PROGRAM MAIN
VAR
	//Main Terminal INPUTS
		//Part 1(Conveyor 1)	
	Inp_Part_at_Conveyor_1								AT%I*: BOOL;
	Inp_Plunger_Parts_Container_In						AT%I*: BOOL;
	Inp_Plunger_Parts_Container_Out						AT%I*: BOOL;
	Inp_Part_On_Conveyor_1								AT%I*: BOOL;
	Inp_Part_in_front_of_Parts_Alignment				AT%I*: BOOL;
	Inp_Plunger_Parts_Alignment_Left_In					AT%I*: BOOL;
	Inp_Plunger_Parts_Alignment_Left_Out				AT%I*: BOOL;
	Inp_Plunger_Parts_Alignment_Right_In				AT%I*: BOOL;	
	
	Inp_Plunger_Parts_Alignment_Right_Out				AT%I*: BOOL;
	Inp_Plunger_Parts_Alignment_Above_In				AT%I*: BOOL;
	Inp_Plunger_Parts_Alignment_Above_Out				AT%I*: BOOL;
	Inp_Part_in_front_of_Crane							AT%I*: BOOL;
	Inp_Crane_In										AT%I*: BOOL;
	Inp_Crane_Out										AT%I*: BOOL;
	Inp_Crane_Above										AT%I*: BOOL;
	Inp_Crane_Below										AT%I*: BOOL;
	
	Inp_Motor_1_Protection_Switch_is_OK					AT%I*: BOOL;
	Inp_Base_Positions									AT%I*: BOOL;
	Inp_Start_Button									AT%I*: BOOL;
	Inp_Stop_Button										AT%I*: BOOL;
	
		//Part 2(Conveyor 2)	
	Inp_Conveyor_2_Palette_Left_Side					AT%I*: BOOL;
	Inp_Conveyor_2_Palette_Right_Side					AT%I*: BOOL;
	Inp_Palette_in_front_of_Tester						AT%I*: BOOL;
	Inp_Stopper_Below									AT%I*: BOOL;
	Inp_Stopper_Above									AT%I*: BOOL;
	Inp_Feedback_from_Tester							AT%I*: BOOL;
	Inp_Reserve_1										AT%I*: BOOL;
	Inp_Motor_2_Protection_Switch_is_OK					AT%I*: BOOL;
	
	Inp_Conveyor_2_Pallete_Slider_In					AT%I*: BOOL;
	Inp_Conveyor_2_Pallete_Slider_Out					AT%I*: BOOL;
	Inp_Feedback_from_Tester_GOOD_Part					AT%I*: BOOL;
	Inp_Feedback_from_Tester_BAD_Part					AT%I*: BOOL;
		
		//Part 3(Conveyor 3)
	Inp_Conveyor_3_Palette_Left_Side					AT%I*: BOOL;
	Inp_Conveyor_3_Palette_Right_Side					AT%I*: BOOL;	
	Inp_Conveyor_3_Pallete_Slider_In					AT%I*: BOOL;
	Inp_Conveyor_3_Pallete_Slider_Out					AT%I*: BOOL;	
	Inp_Motor_3_Protection_Switch_is_OK					AT%I*: BOOL;

	//Coupler	
		//Part 4(Sorting System)
	Inp_Sorter_in_Basik_Position						AT%I*: BOOL;
	Inp_Sorter_Plunger_Above							AT%I*: BOOL;
	Inp_Sorter_Plunger_Below							AT%I*: BOOL;
	Inp_Measuring_Bar_Sorting_Axis_X					AT%I*: INT;
	Inp_Measuring_Bar_Sorting_Axis_Y					AT%I*: INT;
	Inp_Form_is_Changed_Button							AT%I*: BOOL;
	

	//Main Terminal OUTPUTS
		//Part 1(Conveyor 1)	
	Out_Conveyor_1_Motor_On								AT%Q*: BOOL;
	Out_Plunger_Parts_Container_Drive_In				AT%Q*: BOOL;
	Out_Plunger_Parts_Container_Drive_Out				AT%Q*: BOOL;
	Out_Plunger_Parts_Alignment_Left_Drive_In			AT%Q*: BOOL;
	Out_Plunger_Parts_Alignment_Left_Drive_Out			AT%Q*: BOOL;
	Out_Plunger_Parts_Alignment_Right_Drive_In			AT%Q*: BOOL;		
	Out_Plunger_Parts_Alignment_Right_Drive_Out			AT%Q*: BOOL;
	Out_Plunger_Parts_Alignment_Above_Drive_In			AT%Q*: BOOL;
	
	Out_Plunger_Parts_Alignment_Above_Drive_Out			AT%Q*: BOOL;
	Out_Crane_Drive_In									AT%Q*: BOOL;
	Out_Crane_Drive_Out									AT%Q*: BOOL;
	Out_Crane_Drive_Up									AT%Q*: BOOL;
	Out_Crane_Drive_Down								AT%Q*: BOOL;
	
		//Part 2(Conveyor 2)	
	Out_Conveyor_2_Motor_On								AT%Q*: BOOL;
	Out_Stopper_Drive_Up								AT%Q*: BOOL;
	Out_Stopper_Drive_Down								AT%Q*: BOOL;
	Out_Conveyor_2_Pallete_Slider_Drive_In				AT%Q*: BOOL;
	Out_Conveyor_2_Pallete_Slider_Drive_Out				AT%Q*: BOOL;
	
		//Part 3(Conveyor 3)
	Out_Conveyor_3_Motor_On								AT%Q*: BOOL;	
	Out_Conveyor_3_Pallete_Slider_Drive_In				AT%Q*: BOOL;
	Out_Conveyor_3_Pallete_Slider_Drive_Out				AT%Q*: BOOL;

	//Coupler	
		//Part 4(Sorting System)
	Out_Sortierer_Pluger_Drive_Up						AT%Q*: BOOL;
	Out_Sortierer_Pluger_Drive_Down						AT%Q*: BOOL;	
	Out_Measuring_Bar_Sorting_Axis_X_Motor_On			AT%Q*: BOOL;
	Out_Measuring_Bar_Sorting_Axis_Y_Motor_On			AT%Q*: BOOL;
	Out_Sorter_Pluger_Pull_in							AT%Q*: BOOL;
	
	position:Positions;
	a:INT;
	motor_Sorting:Motor_Sorting;
	conveyor_1:Conveyor_1;
	conveyor_2:Conveyor_2;
	conveyor_3:Conveyor_3;
	Buffer_VAR_Feedback_from_Tester_GOOD_Part:BOOL;
	Buffer_VAR_Feedback_from_Tester_BAD_Part:BOOL;
	M_Machine_Release										: RS;
	Machine_Base_Position:Machine_Base_Position;
END_VAR

M_Machine_Release(
SET:= Inp_Start_Button AND Machine_Base_Position.BOOL_Base_Position, 
RESET1:= Inp_Stop_Button);

motor_Sorting(
	Inp_Conveyor_2_Palette_Right_Side_at_Sorter:= , 
	Inp_Sortierer_in_Basic_Position:= , 
	Inp_Sorter_Plunger_Above:= , 
	Inp_Sorter_Plunger_Below:= , 
	Inp_Measuring_Bar_Sorting_Axis_X:= , 
	Inp_Measuring_Bar_Sorting_Axis_Y:= , 
	Inp_Form_is_Changed_Button:= , 
	Out_Sorter_Pluger_Drive_Up=> , 
	BOOL_Feedback_from_Tester_GOOD_Part:= Buffer_VAR_Feedback_from_Tester_GOOD_Part, 
	BOOL_Feedback_from_Tester_BAD_Part:= Buffer_VAR_Feedback_from_Tester_BAD_Part, 
	Out_Sorter_Pluger_Drive_Down=> , 
	Out_Measuring_Bar_Sorting_Axis_X_Right_Rotation_Motor_On=> , 
	Out_Measuring_Bar_Sorting_Axis_Y_Right_Rotation_Motor_On=> , 
	Out_Measuring_Bar_Sorting_Axis_X_Left_Rotation_Motor_On=> , 
	Out_Measuring_Bar_Sorting_Axis_Y_Left_Rotation_Motor_On=> , 
	Out_Sorter_Pluger_Pull_in=> , 
	Palette_at_Sorter_is_free=> );
	
	conveyor_1(
	Inp_Part_at_Conveyor_1:= Inp_Part_at_Conveyor_1, 
	Inp_Plunger_Parts_Container_In:= Inp_Plunger_Parts_Container_In, 
	Inp_Plunger_Parts_Container_Out:= Inp_Plunger_Parts_Container_Out, 
	Inp_Part_On_Conveyor_1:= Inp_Part_On_Conveyor_1, 
	Inp_Part_in_front_of_Parts_Alignment:= Inp_Part_in_front_of_Parts_Alignment, 
	Inp_Plunger_Parts_Alignment_Left_In:= Inp_Plunger_Parts_Alignment_Left_In, 
	Inp_Plunger_Parts_Alignment_Left_Out:= Inp_Plunger_Parts_Alignment_Left_Out, 
	Inp_Plunger_Parts_Alignment_Right_In:= Inp_Plunger_Parts_Alignment_Right_In, 
	Inp_Plunger_Parts_Alignment_Right_Out:= Inp_Plunger_Parts_Alignment_Right_Out, 
	Inp_Plunger_Parts_Alignment_Above_In:= Inp_Plunger_Parts_Alignment_Above_In, 
	Inp_Plunger_Parts_Alignment_Above_Out:= Inp_Plunger_Parts_Alignment_Above_Out, 
	Inp_Part_in_front_of_Crane:= Inp_Part_in_front_of_Crane, 
	Inp_Crane_In:= Inp_Crane_In, 
	Inp_Crane_Out:= Inp_Crane_Out, 
	Inp_Crane_Above:= Inp_Crane_Above, 
	Inp_Crane_Below:= Inp_Crane_Below, 
	Inp_Motor_1_Protection_Switch_is_OK:= Inp_Motor_1_Protection_Switch_is_OK, 
	Inp_Base_Positions:= Inp_Base_Positions, 
	Out_Conveyor_1_Motor_On=> , 
	Out_Plunger_Parts_Container_Drive_In=> , 
	Out_Plunger_Parts_Container_Drive_Out=> , 
	Out_Plunger_Parts_Alignment_Left_Drive_In=> , 
	Out_Plunger_Parts_Alignment_Left_Drive_Out=> , 
	Out_Plunger_Parts_Alignment_Right_Drive_In=> , 
	Out_Plunger_Parts_Alignment_Right_Drive_Out=> , 
	Out_Plunger_Parts_Alignment_Above_Drive_In=> , 
	Out_Plunger_Parts_Alignment_Above_Drive_Out=> , 
	Out_Crane_Drive_In=> , 
	Out_Crane_Drive_Out=> , 
	Out_Crane_Drive_Up=> , 
	Out_Crane_Drive_Down=> , 
	Out_Crane_Take_a_Part=> , 
	M_Part_is_shipped_on_the_Conveyor_2=> );
	
	conveyor_2(
	Inp_Conveyor_2_Palette_Left_Side:= Inp_Conveyor_2_Palette_Left_Side, 
	Inp_Conveyor_2_Palette_Right_Side:= Inp_Conveyor_2_Palette_Right_Side, 
	Inp_Palette_in_front_of_Tester:= Inp_Palette_in_front_of_Tester, 
	Inp_Stopper_Below:= Inp_Stopper_Below, 
	Inp_Stopper_Above:= Inp_Stopper_Above, 
	BOOL_Feedback_from_Tester_GOOD_Part:= Buffer_VAR_Feedback_from_Tester_GOOD_Part, 
	BOOL_Feedback_from_Tester_BAD_Part:= Buffer_VAR_Feedback_from_Tester_BAD_Part, 
	Inp_Motor_2_Protection_Switch_is_OK:= Inp_Motor_2_Protection_Switch_is_OK, 
	Inp_Conveyor_2_Pallete_Slider_In:= Inp_Conveyor_2_Pallete_Slider_In, 
	Inp_Conveyor_2_Pallete_Slider_Out:= Inp_Conveyor_2_Pallete_Slider_Out, 
	Out_Conveyor_2_Motor_On=> , 
	Out_Stopper_Drive_Up=> , 
	Out_Stopper_Drive_Down=> , 
	Out_Conveyor_2_Pallete_Slider_Drive_In=> , 
	Out_Conveyor_2_Pallete_Slider_Drive_Out=> , 
	M_Conveyor_2_is_ready_to_take_Part_From_Conveyor_2=> , 
	M_Part_is_ready_for_Test=> );
	
	conveyor_3(
	Inp_Conveyor_3_Palette_Left_Side:= Inp_Conveyor_3_Palette_Left_Side, 
	Inp_Conveyor_3_Palette_Right_Side:= Inp_Conveyor_3_Palette_Right_Side, 
	Inp_Conveyor_3_Pallete_Slider_In:= Inp_Conveyor_3_Pallete_Slider_In, 
	Inp_Conveyor_3_Pallete_Slider_Out:= Inp_Conveyor_3_Pallete_Slider_Out, 
	Inp_Motor_3_Protection_Switch_is_OK:= Inp_Motor_3_Protection_Switch_is_OK, 
	Inp_Conveyor_2_Palette_Right_Side:= Inp_Conveyor_2_Palette_Right_Side, 
	Out_Conveyor_3_Motor_On=> , 
	Out_Conveyor_3_Pallete_Slider_Drive_In=> , 
	Out_Conveyor_3_Pallete_Slider_Drive_Out=> ,
	Out_Sortierer_Pluger_Drive_Up=> , 
	Out_Sortierer_Pluger_Drive_Down=> , 
	Out_Measuring_Bar_Sorting_Axis_X_Motor_On=> , 
	Out_Measuring_Bar_Sorting_Axis_Y_Motor_On=> , 
	Out_Sorter_Pluger_Pull_in=> );
	
	Machine_Base_Position(
	Inp_Base_Positions:= Inp_Base_Positions );
	
	IF Inp_Feedback_from_Tester_GOOD_Part OR Main.motor_Sorting.Write_BOOL_Feedback_from_Tester_GOOD_Part
		THEN Buffer_VAR_Feedback_from_Tester_GOOD_Part:=TRUE;
	END_IF
		IF Inp_Feedback_from_Tester_GOOD_Part=FALSE OR Main.motor_Sorting.Write_BOOL_Feedback_from_Tester_GOOD_Part=FALSE
		THEN Buffer_VAR_Feedback_from_Tester_GOOD_Part:=FALSE;
	END_IF
	
		IF Inp_Feedback_from_Tester_BAD_Part OR Main.motor_Sorting.Write_BOOL_Feedback_from_Tester_BAD_Part
		THEN Buffer_VAR_Feedback_from_Tester_BAD_Part:=TRUE;
	END_IF
		IF Inp_Feedback_from_Tester_BAD_Part=FALSE OR Main.motor_Sorting.Write_BOOL_Feedback_from_Tester_BAD_Part=FALSE
		THEN Buffer_VAR_Feedback_from_Tester_BAD_Part:=FALSE;
	END_IF

END_PROGRAM

(* stored: Version 1.1.0.1, ProductVersion 3.1.4024.12
   POU MAIN: Id {963367b4-7853-46d9-a119-421c43f5684c}, SpecialFunc None *)
